// TIA Portal V17 export
// export: Created 2023-02-14T02:49:54.8498905Z, ExportSetting WithDefaults, DisplayName Totally Integrated Automation Portal, DisplayVersion V17, DisplayName TIA Portal Openness, DisplayVersion V17, DisplayName TIA Portal Teamcenter Gateway, DisplayVersion V17, DisplayName TIA Portal Version Control Interface, DisplayVersion V17, DisplayName SINAMICS Startdrive Advanced, DisplayVersion V17, DisplayName SINAMICS Startdrive G130, G150, S120, S150, SINAMICS MV, S210, DisplayVersion V17, DisplayName SINAMICS Startdrive G110M, G120, G120C, G120D, G120P, G115D, DisplayVersion V17, DisplayName STEP 7 Professional, DisplayVersion V17, DisplayName STEP 7 Safety, DisplayVersion V17, DisplayName WinCC Professional, DisplayVersion V17
VAR_GLOBAL   // PLC tag table "RIO MCC Preparation"
   "P-02.01 SW" AT %IW912 : Word;
   "P-02.01 AV" AT %IW914 : Int;
   "P-02.01 Voltage" AT %IW916 : Int;
   "P-02.01 Ampere" AT %IW918 : Int;
   "P-02.01 KW" AT %IW920 : Int;
   "P-02.01 Nm" AT %IW922 : Int;
   "P-02.03 SW" AT %IW924 : Word;
   "P-02.03 AV" AT %IW926 : Int;
   "P-02.03 Voltage" AT %IW928 : Int;
   "P-02.03 Ampere" AT %IW930 : Int;
   "P-02.03 KW" AT %IW932 : Int;
   "P-02.03 Nm" AT %IW934 : Int;
   "P-03.01 SW" AT %IW936 : Word;
   "P-03.01 AV" AT %IW938 : Int;
   "P-03.01 Voltage" AT %IW940 : Int;
   "P-03.01 Ampere" AT %IW942 : Int;
   "P-03.01 KW" AT %IW944 : Int;
   "P-03.01 Nm" AT %IW946 : Int;
   "P-03.03 SW" AT %IW948 : Word;
   "P-03.03 AV" AT %IW950 : Int;
   "P-03.03 Voltage" AT %IW952 : Int;
   "P-03.03 Ampere" AT %IW954 : Int;
   "P-03.03 KW" AT %IW956 : Int;
   "P-03.03 Nm" AT %IW958 : Int;
   "P-04.01 SW" AT %IW960 : Word;
   "P-04.01 AV" AT %IW962 : Int;
   "P-04.01 Voltage" AT %IW964 : Int;
   "P-04.01 Ampere" AT %IW966 : Int;
   "P-04.01 KW" AT %IW968 : Int;
   "P-04.01 Nm" AT %IW970 : Int;
   "XA-05.01 SW" AT %IW984 : Word;
   "XA-05.01 AV" AT %IW986 : Int;
   "XA-05.01 Voltage" AT %IW988 : Int;
   "XA-05.01 Ampere" AT %IW990 : Int;
   "XA-05.01 KW" AT %IW992 : Int;
   "XA-05.01 Nm" AT %IW994 : Int;
   "P-05.01 SW" AT %IW996 : Word;
   "P-05.01 AV" AT %IW998 : Int;
   "P-05.01 Voltage" AT %IW1000 : Int;
   "P-05.01 Ampere" AT %IW1002 : Int;
   "P-05.01 KW" AT %IW1004 : Int;
   "P-05.01 Nm" AT %IW1006 : Int;
   "P-06.01 SW" AT %IW1008 : Word;
   "P-06.01 AV" AT %IW1010 : Int;
   "P-06.01 Voltage" AT %IW1012 : Int;
   "P-06.01 Ampere" AT %IW1014 : Int;
   "P-06.01 KW" AT %IW1016 : Int;
   "P-06.01 Nm" AT %IW1018 : Int;
   "P-07.01 SW" AT %IW1020 : Word;
   "P-07.01 AV" AT %IW1022 : Int;
   "P-07.01 Voltage" AT %IW1024 : Int;
   "P-07.01 Ampere" AT %IW1026 : Int;
   "P-07.01 KW" AT %IW1028 : Int;
   "P-07.01 Nm" AT %IW1030 : Int;
   "P-08.01 SW" AT %IW1032 : Word;
   "P-08.01 AV" AT %IW1034 : Int;
   "P-08.01 Voltage" AT %IW1036 : Int;
   "P-08.01 Ampere" AT %IW1038 : Int;
   "P-08.01 KW" AT %IW1040 : Int;
   "P-08.01 Nm" AT %IW1042 : Int;
   "XA-09.01 SW" AT %IW1044 : Word;
   "XA-09.01 AV" AT %IW1046 : Int;
   "XA-09.01 Voltage" AT %IW1048 : Int;
   "XA-09.01 Ampere" AT %IW1050 : Int;
   "XA-09.01 KW" AT %IW1052 : Int;
   "XA-09.01 Nm" AT %IW1054 : Int;
   "P-09.01 SW" AT %IW1056 : Word;
   "P-09.01 AV" AT %IW1058 : Int;
   "P-09.01 Voltage" AT %IW1060 : Int;
   "P-09.01 Ampere" AT %IW1062 : Int;
   "P-09.01 KW" AT %IW1064 : Int;
   "P-09.01 Nm" AT %IW1066 : Int;
   "P-10.01 SW" AT %IW1068 : Word;
   "P-10.01 AV" AT %IW1070 : Int;
   "P-10.01 Voltage" AT %IW1072 : Int;
   "P-10.01 Ampere" AT %IW1074 : Int;
   "P-10.01 KW" AT %IW1076 : Int;
   "P-10.01 Nm" AT %IW1078 : Int;
   "P-51.01 Alarm" AT %I69.0 : Bool;
   "P-05.03 Overload" AT %I69.1 : Bool;
   "P-08.02 Alarm" AT %I69.2 : Bool;
   "P-09.03 Overload" AT %I69.3 : Bool;
   "P-51.01  Feedback" AT %I69.4 : Bool;
   "P-05.03  Feedback" AT %I69.5 : Bool;
   "P-08.02  Feedback" AT %I69.6 : Bool;
   "P-09.03  Feedback" AT %I69.7 : Bool;
   "Emergency Stop MCC Preparation" AT %I70.0 : Bool;
   "MCC Prep Spare 2" AT %I70.1 : Bool;
   "MCC Prep Spare 3" AT %I70.2 : Bool;
   "MCC Prep Spare 4" AT %I70.3 : Bool;
   "MCC Prep Spare 5" AT %I70.4 : Bool;
   "MCC Prep Spare 6" AT %I70.5 : Bool;
   "MCC Prep Spare 7" AT %I70.6 : Bool;
   "MCC Prep Spare 8" AT %I70.7 : Bool;
   "P-51.01 Act" AT %IW676 : Int;
   "P-08.02 Act" AT %IW678 : Int;
   "MCC Prep Spare 13" AT %IW680 : Int;
   "MCC Prep Spare 14" AT %IW682 : Int;
   "Start/Stop P-51.01" AT %Q6.0 : Bool;
   "Start/Stop P-05.03" AT %Q6.1 : Bool;
   "Start/Stop P-08.02" AT %Q6.2 : Bool;
   "Start/Stop P-09.03" AT %Q6.3 : Bool;
   "P-02.01 CW" AT %QW912 : Word;
   "P-02.01 SP" AT %QW914 : Word;
   "P-02.03 CW" AT %QW924 : Word;
   "P-02.03 SP" AT %QW926 : Word;
   "P-03.01 CW" AT %QW936 : Word;
   "P-03.01 SP" AT %QW938 : Word;
   "P-03.03 CW" AT %QW948 : Word;
   "P-03.03 SP" AT %QW950 : Word;
   "P-04.01 CW" AT %QW960 : Word;
   "P-04.01 SP" AT %QW962 : Word;
   "XA-05.01 CW" AT %QW984 : Word;
   "XA-05.01 SP" AT %QW986 : Word;
   "P-05.01 CW" AT %QW996 : Word;
   "P-05.01 SP" AT %QW998 : Word;
   "P-06.01 CW" AT %QW1008 : Word;
   "P-06.01 SP" AT %QW1010 : Word;
   "P-07.01 CW" AT %QW1020 : Word;
   "P-07.01 SP" AT %QW1022 : Word;
   "P-08.01 CW" AT %QW1032 : Word;
   "P-08.01 SP" AT %QW1034 : Word;
   "XA-09.01 CW" AT %QW1044 : Word;
   "XA-09.01 SP" AT %QW1046 : Word;
   "P-09.01 CW" AT %QW1056 : Word;
   "P-09.01 SP" AT %QW1058 : Word;
   "P-10.01 CW" AT %QW1068 : Word;
   "P-10.01 SP" AT %QW1070 : Word;
   "MCC Prep Spare 9" AT %Q6.4 : Bool;
   "P-51.01 SP" AT %QW74 : Int;
   "P-08.02 SP" AT %QW76 : Int;
   "MCC Prep Spare 10" AT %Q6.5 : Bool;
   "MCC Prep Spare 11" AT %Q6.6 : Bool;
   "MCC Prep Spare 12" AT %Q6.7 : Bool;
   "MCC Prep Spare 15" AT %QW78 : Int;
   "MCC Prep Spare 16" AT %QW80 : Int;
   "P-05.03 SW" AT %MW80 : Word;   // Temporary address
   "P-05.03 AV" AT %MW82 : Word;   // Temporary address
   "P-05.03 Voltage" AT %MW84 : Word;   // Temporary address
   "P-05.03 Ampere" AT %MW86 : Word;   // Temporary address
   "P-05.03 KW" AT %MW88 : Word;   // Temporary address
   "P-05.03 Nm" AT %MW90 : Word;   // Temporary address
   "P-05.03 CW" AT %MW92 : Word;   // Temporary address
   "P-05.03 SP" AT %MW94 : Word;   // Temporary address
END_VAR
